Staubli VAL3: getDetectDist.pgx

program getDetectDist(num x_nConvNum (dimensions=1), num x_nIdx (dimensions=1), num& x_nDetectDist[] (dimensions=1), num& x_nError[] (dimensions=1))
  local point l_pDummy
  local point l_pPoint
begin
  // This program return the distance in between the detection
  // device and the frame of the conveyor
  //
  // Input param
  //  x_nIdx  : Index of the object in the queue
  //
  // Output param
  //  x_nDetectDist : Distance
  //  x_nError: Error code
  //    0 : No error
  //    1 : No object selected
  //    2 : Object with requested ID has not been calibrated
  //
  //----------------------------------------------------------------
  //
  //
  switch x_nConvNum
    case 0
      call cnv0:getDetectDist(x_nIdx,x_nDetectDist,x_nError)
    break
    case 1
      call cnv1:getDetectDist(x_nIdx,x_nDetectDist,x_nError)
    break
  endSwitch
end
